PROGRAM P_FeedForward
VAR
	
	fbFFOne : FB_FeedForward;
	fbFFTwo : FB_FeedForward;
	
END_VAR


fbFFOne(
	fPs := G_OPC.fPs.fDanielFilter,
	fPa := G_OPC.fMainPaDCV.fDanielFilter,
	fPb := G_OPC.fMainPbDCV.fDanielFilter,
	
	fXDot := G_OPC.fXDotRefOne,
	fDeltaP0 := G_Parameters.fDeltaP0One,
	
	fMaxFlowUp := G_Parameters.fQMaxUpOne,
	fMaxFlowDown := G_Parameters.fQMaxUpOne,
	
	fDeadBandUp := G_Parameters.fDeadUpOne,
	fDeadBandDown := G_Parameters.fDeadDownOne,
	
	fArea := G_Parameters.fAreaOne,
	fPhi := G_Parameters.fAreaRelationOne,
	
	fUFF => G_OPC.fValveOneSignals.fFF
);

fbFFTwo(
	fPs := G_OPC.fPs.fDanielFilter,
	fPa := G_OPC.fJibPaDCV.fDanielFilter,
	fPb := G_OPC.fJibPbDCV.fDanielFilter,
	
	fXDot := G_OPC.fXDotRefTwo,
	fDeltaP0 := G_Parameters.fDeltaP0Two,
	
	fMaxFlowUp := G_Parameters.fQMaxUpTwo,
	fMaxFlowDown := G_Parameters.fQMaxUpTwo,
	
	fDeadBandUp := G_Parameters.fDeadUpTwo,
	fDeadBandDown := G_Parameters.fDeadDownTwo,
	
	fArea := G_Parameters.fAreaTwo,
	fPhi := G_Parameters.fAreaRelationTwo,
	
	fUFF => G_OPC.fValveTwoSignals.fFF
);

END_PROGRAM

(* stored: Version 1.1.0.1
   POU P_FeedForward: Id {27679076-0387-4864-af79-9c330260a68e}, SpecialFunc None *)
